TYPE ST_HMI_PowerMeas :
STRUCT
	Voltage			: REAL;
	Frequency		: REAL;
	ActivePower		: REAL;
	ReactivePower	: REAL;
	Current			: REAL;
END_STRUCT
END_TYPE

(* stored: Version 1.1.0.1, ProductVersion 3.1.4026.18
   DUT ST_HMI_PowerMeas: Id {d0175068-27c9-4e46-bde8-44a821dbd064} *)
